// TIA Portal V17 export
// export: Created 2025-03-10T13:09:23.9602692Z, ExportSetting WithDefaults, DisplayName Totally Integrated Automation Portal, DisplayVersion V17 Update 8, DisplayName TIA Portal Openness, DisplayVersion V17 Update 8, DisplayName TIA Portal Version Control Interface, DisplayVersion V17, DisplayName SINAMICS Startdrive Advanced, DisplayVersion V17 SP2, DisplayName SINAMICS Startdrive G110M, G120, G120C, G120D, G120P, G115D, DisplayVersion V17 SP2, DisplayName SINAMICS Startdrive G130, G150, S120, S150, SINAMICS MV, S210, DisplayVersion V17 SP2, DisplayName STEP 7 Professional, DisplayVersion V17 Update 8, DisplayName SINUMERIK ONE STEP 7 Toolbox, DisplayVersion V17 Update 12, DisplayName SINUMERIK 840D sl STEP 7 Toolbox, DisplayVersion V17 Update 12, DisplayName STEP 7 Safety, DisplayVersion V17 Update 6, DisplayName WinCC Advanced, DisplayVersion V17 Update 8
DATA_BLOCK "LBP_MFuncDecListConfig"   // DB75
TITLE = M decoding acc. to list / Decodificación M seg. lista / M-Decodierung gem. Liste
{ S7_Optimized_Access := 'FALSE'; DB_Accessible_From_OPC_UA := 'FALSE' }
AUTHOR : SINUMERIK
FAMILY : SINUMERIK_ONE
VERSION : 6.15
// Interface between user program and NCK, contains the configuration for the M functions to be decoded / Interfaz entre programa de usuario y NCK, contiene la configuración para las funciones M que deben decodificarse. / Schnittstelle zwischen Anwenderprogramm und NCK, enthält die Konfiguration für die zu decodierenden M-Funktionen
// stored: AutoNumber false, DBAccessibleFromOPCUA false, DBAccessibleFromWebserver true, IsOnlyStoredInLoadMemory false, IsWriteProtectedInAS false
   VAR RETAIN
      MSigGrp : Array[1..16] of Struct
         MExtAdr : Int;
         MFirstAdr : DInt;
         MLastAdr : DInt;
      END_STRUCT;
   END_VAR
BEGIN
   MSigGrp[1..16].MFirstAdr := DINT#0;
   MSigGrp[1..16].MLastAdr := DINT#0;
END_DATA_BLOCK
